TYPE ST_MarkState :
STRUCT
  bSet        : BOOL;     // mark was set (detected)
  bMissed     : BOOL;     // mark was missing (+internally generated)
  bInArea     : BOOL;     // mark withing ok area
  dx          : LREAL;    // x displacement [m]
  dy          : LREAL;    // y displacement [m]
  fLengthReal : LREAL;    // real detected mark length [m]
  nPosXReal   : DINT;     // detected position X absolute [SubPx]
  END_STRUCT
END_TYPE

(* stored: Version 1.1.0.1, ProductVersion 3.1.4024.11
   DUT ST_MarkState: Id {3261b978-bbc5-48eb-82c2-091ced97e2f3} *)
